TYPE InterlockState :
STRUCT
	aLogicalInterlock				: ARRAY[1..GVL_CONSTANT.NumLogicalInterlockState] OF BOOL;
	aInterlockSubstate				: LogicalInterlockSubstate;
	aAlarmState						: ARRAY[1..GVL_CONSTANT.NumInterlockAlarmWarningState] OF BOOL;
	aWarningState					: ARRAY[1..GVL_CONSTANT.NumInterlockAlarmWarningState] OF BOOL;
END_STRUCT
END_TYPE

(* stored: Version 1.1.0.1, ProductVersion 3.1.4026.11
   DUT InterlockState: Id {ae594bee-db28-4782-9cde-bc0fe5f8df3e} *)
